FUNCTION_BLOCK NeredaDAeration (* Composite Function Block Type *)
  (* Standard: 61499-2 *)
  (* Version 0.0, 4/25/2024, SESA713705, Schneider Electric, template *)
  PACKAGE SE.Nereda;
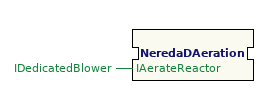
  SOCKETS
    IAerateReactor : IDedicatedBlower;
  END_SOCKETS
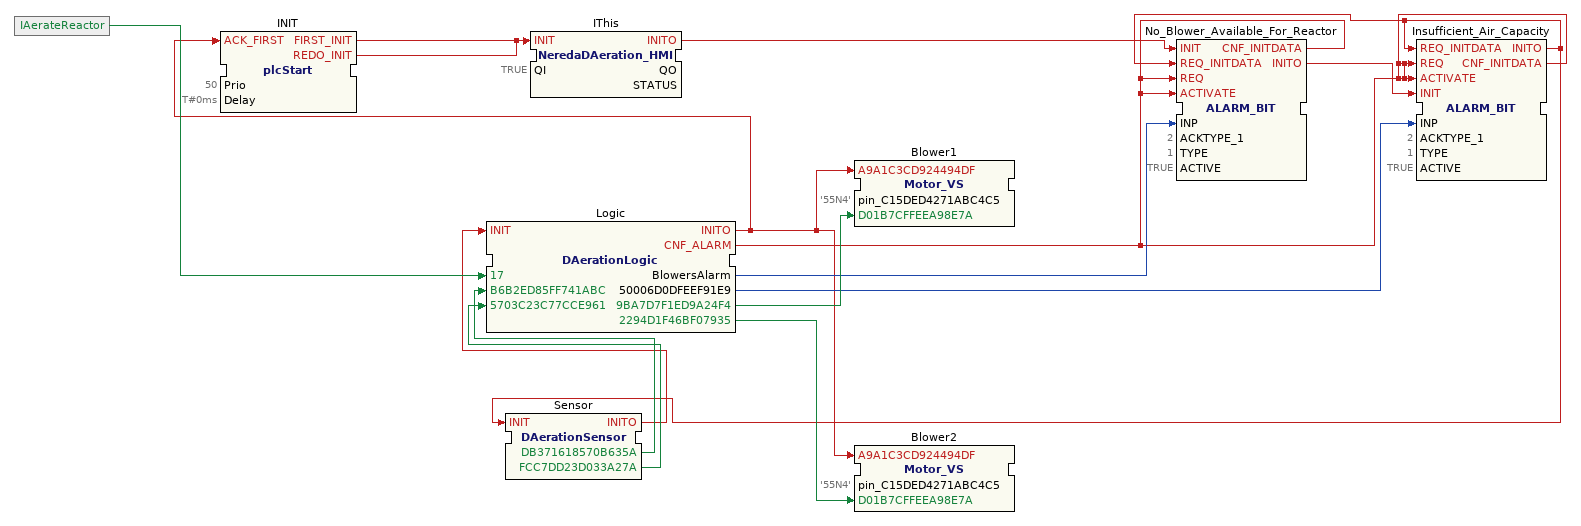
  (* 01 - FUNCTIONNAL INPUT INTERFACE *)
  (* 00 - INITIALIZATION *)
  (* 05 - LOGIC *)
  (* 06 - HMI INTERFACE *)
  (* 03 - FIELD INTERFACE *)
  (* 02 - FUNCTIONNAL OUTPUT INTERFACE *)
  (* Aeartion Logic *)
  (* 04 - CHILDREN *)
  (* 4A - TYPICALS *)
  (* 07- REACTOR ALARM *)
  FBS
    Logic : DAerationLogic;
    IThis : NeredaDAeration_HMI(QI := TRUE);
    INIT : plcStart(Prio := 50, Delay := T#0ms);
    Sensor : DAerationSensor;
    No_Blower_Available_For_Reactor : ALARM_BIT(ACKTYPE_1 := 2, TYPE := 1, ACTIVE := TRUE);
    Blower1 : Motor_VS(pin_C15DED4271ABC4C5 := '55N4');
    Blower2 : Motor_VS(pin_C15DED4271ABC4C5 := '55N4');
    Insufficient_Air_Capacity : ALARM_BIT(ACKTYPE_1 := 2, TYPE := 1, ACTIVE := TRUE);
  END_FBS
  EVENT_CONNECTIONS
    INIT.FIRST_INIT TO IThis.INIT;
    IThis.INITO TO No_Blower_Available_For_Reactor.INIT;
    Insufficient_Air_Capacity.INITO TO No_Blower_Available_For_Reactor.REQ_INITDATA;
    No_Blower_Available_For_Reactor.CNF_INITDATA TO No_Blower_Available_For_Reactor.REQ;
    INIT.REDO_INIT TO IThis.INIT;
    No_Blower_Available_For_Reactor.CNF_INITDATA TO No_Blower_Available_For_Reactor.ACTIVATE;
    Insufficient_Air_Capacity.INITO TO Sensor.INIT;
    Sensor.INITO TO Logic.INIT;
    Logic.INITO TO INIT.ACK_FIRST;
    Logic.INITO TO Blower1.A9A1C3CD924494DF;
    Logic.INITO TO Blower2.A9A1C3CD924494DF;
    Logic.CNF_ALARM TO No_Blower_Available_For_Reactor.REQ;
    Insufficient_Air_Capacity.INITO TO Insufficient_Air_Capacity.REQ_INITDATA;
    Insufficient_Air_Capacity.CNF_INITDATA TO Insufficient_Air_Capacity.REQ;
    Insufficient_Air_Capacity.CNF_INITDATA TO Insufficient_Air_Capacity.ACTIVATE;
    No_Blower_Available_For_Reactor.INITO TO Insufficient_Air_Capacity.INIT;
    Logic.CNF_ALARM TO Insufficient_Air_Capacity.REQ;
  END_CONNECTIONS
  DATA_CONNECTIONS
    Logic.BlowersAlarm TO No_Blower_Available_For_Reactor.INP;
    Logic.50006D0DFEEF91E9 TO Insufficient_Air_Capacity.INP;
  END_CONNECTIONS
  ADAPTER_CONNECTIONS
    Logic.9BA7D7F1ED9A24F4 TO Blower1.D01B7CFFEEA98E7A;
    Logic.2294D1F46BF07935 TO Blower2.D01B7CFFEEA98E7A;
    IAerateReactor TO Logic.17;
    Sensor.DB371618570B635A TO Logic.B6B2ED85FF741ABC;
    Sensor.FCC7DD23D033A27A TO Logic.5703C23C77CCE961;
  END_CONNECTIONS
END_FUNCTION_BLOCK
